INTERFACE ITF_SubsystemTransport EXTENDS __System.IQueryInterface

METHOD M_CallInterface : BOOL
VAR_IN_OUT
	mErrorData				: ST_ErrorDataSet; // Error data
END_VAR
END_METHOD

METHOD M_GetTransportData : REFERENCE TO ST_TransportData
END_METHOD

METHOD M_Init : BOOL
VAR_INPUT
	mInit			: BOOL; // Force init
END_VAR
END_METHOD

METHOD M_MoveTU_DataIndex : DINT
END_METHOD

END_INTERFACE

(* stored: Version 1.1.0.1, ProductVersion 3.1.4022.12
   Itf ITF_SubsystemTransport: Id {a187486f-7e82-4244-b5a8-da5e63f23146}
   Method M_CallInterface: Id {e36329f5-62e4-4c67-8d16-7de249df4d87}
   Method M_GetTransportData: Id {924d7631-b4c2-48fa-9a98-c587bed4b0aa}
   Method M_Init: Id {a1328f45-e491-4711-9268-d39463679b25}
   Method M_MoveTU_DataIndex: Id {642eaea3-f1e2-40eb-b917-d5d079e62864} *)
